// TIA Portal V17 export
TextList "Codex_TextList_Status"  ListRange=Decimal, Comment="Codex text list import/export loop test."
  TextListEntry   EntryType=SingleValue, Text="停止"
  TextListEntry   EntryType=SingleValue, From=1, To=1, Text="运行"
